// TIA Portal V18 export
FUNCTION_BLOCK "SetA2"   // FB23, FBD
{ S7_Optimized_Access := 'TRUE' }
VERSION : 0.1
// stored: AutoNumber true, IsIECCheckEnabled false, IsRetainMemResEnabled false, MemoryReserve 100, SetENOAutomatically false, UDAEnableTagReadback false
   VAR_INPUT
      xCalibSwMaster : Bool;
      xCalibSwSlave : Bool;
      parMasterCalibPos : Real;
      parSlaveCalibPos : Real;
      btnCopyMasterNow : Bool;
      btnAdjustHorizonPlusStep : Bool;
      btnAdjustHorizonMinusStep : Bool;
      MasterPos : Real;
      SlavePos : Real;
      StepHorAdjust : Real := 10.0;
   END_VAR
   VAR_OUTPUT
      MasterCalibPos : Real;
      MasterCalibNow : Bool;
      SlaveCalibPos : Real;
      SlaveCalibNow : Bool;
   END_VAR
   VAR
      CorrectionFactor : Bool;
      ton { S7_SetPoint := 'True'} : TON_TIME;
      ton1 { S7_SetPoint := 'True'} : TON_TIME;
   END_VAR
BEGIN

REGION Network 1
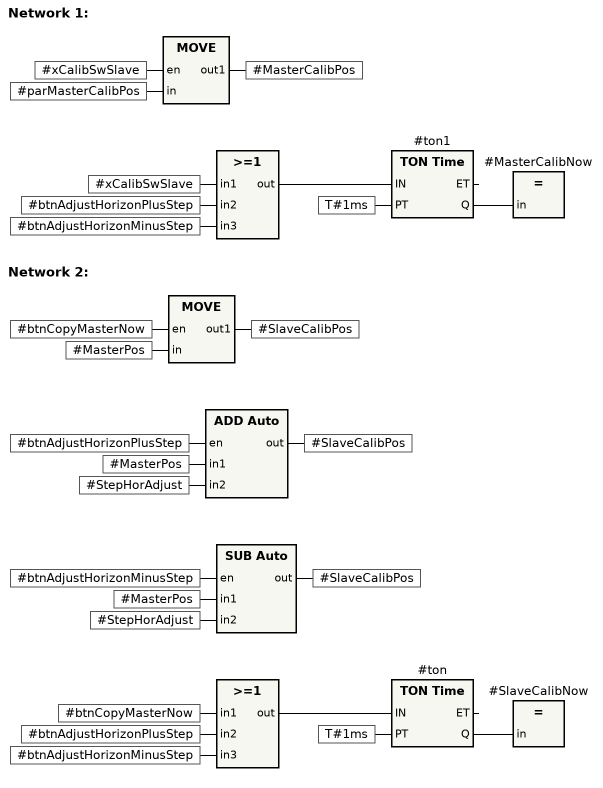
   IF #xCalibSwSlave THEN #MasterCalibPos := #parMasterCalibPos; END_IF;
   #ton1(IN := #xCalibSwSlave OR #btnAdjustHorizonPlusStep OR #btnAdjustHorizonMinusStep, PT := T#1ms);   // TON
   #MasterCalibNow := #ton1.Q;
END_REGION

REGION Network 2
   IF #btnCopyMasterNow THEN #SlaveCalibPos := #MasterPos; END_IF;
   IF #btnAdjustHorizonPlusStep THEN #SlaveCalibPos := #MasterPos + #StepHorAdjust; END_IF;
   IF #btnAdjustHorizonMinusStep THEN #SlaveCalibPos := #MasterPos - #StepHorAdjust; END_IF;
   #ton(IN := #btnCopyMasterNow OR #btnAdjustHorizonPlusStep OR #btnAdjustHorizonMinusStep, PT := T#1ms);   // TON
   #SlaveCalibNow := #ton.Q;
END_REGION
END_FUNCTION_BLOCK
